{attribute 'qualified_only'}
VAR_GLOBAL
	dtCurrentDt : DATE_AND_TIME := DT#2023-02-14-15:24:00;
	tVariable : TIME := T#5S;
END_VAR

(* stored: Version 1.1.0.1, ProductVersion 3.1.4024.12
   GVL GVL_Task1: Id {da98ec69-91f1-4aa5-824a-3b8a4bd16992} *)
